// TIA Portal V17 export
// export: Created 2025-04-09T16:55:10.717677Z, ExportSetting WithDefaults, DisplayName Totally Integrated Automation Portal, DisplayVersion V17, DisplayName TIA Portal Openness, DisplayVersion V17, DisplayName TIA Portal Version Control Interface, DisplayVersion V17, DisplayName STEP 7 Professional, DisplayVersion V17, DisplayName STEP 7 Safety, DisplayVersion V17, DisplayName WinCC Advanced, DisplayVersion V17
VAR_GLOBAL   // PLC tag table "Output"
   Q0 AT %Q22.0 : Bool;
   Q1 AT %Q22.1 : Bool;
   Q2 AT %Q22.2 : Bool;
   Q3 AT %Q22.3 : Bool;
   Q4 AT %Q22.4 : Bool;
   Q5 AT %Q22.5 : Bool;
   Q6 AT %Q22.6 : Bool;
   Q7 AT %Q22.7 : Bool;
   Q8 AT %Q23.0 : Bool;
   Q9 AT %Q23.1 : Bool;
   Q10 AT %Q23.2 : Bool;
   Q11 AT %Q23.3 : Bool;
   Q12 AT %Q23.4 : Bool;
   Q13 AT %Q23.5 : Bool;
   Q14 AT %Q23.6 : Bool;
   Q15 AT %Q23.7 : Bool;
END_VAR
